Fanuc KAREL source: kt00787.KL

-- PROVISIONAL review KL for V940-1; original PC SHA256 72e38fe0c1494964cbfeffb43e855b68a07ae1adb04706cd9a4cfc98baf3447f
-- Incomplete behavior may be omitted. Consult companion uncertainty JSON. Do not deploy.
PROGRAM KT00787
%NOLOCKGROUP
VAR
  R1 : REAL
  R2 : REAL
  OUT : REAL
BEGIN
  -- V9_ZERO_TABLE_METADATA_HINT layout=0001; no indexed target words; source/name/runtime held
  -- UNRESOLVED_PC offsets 5-16; opcodes 2E,23
  -- UNRESOLVED_PC offsets 21-32; opcodes 2E,23
  -- UNRESOLVED_PC offsets 37-48; opcodes 2E,23
  -- UNRESOLVED_PC offsets 53-64; opcodes 2E,23
  -- UNRESOLVED_PC offsets 69-84; opcodes 27,22,76,23
  -- UNRESOLVED_PC offsets 89-93; opcodes 7F
END KT00787
